{attribute 'qualified_only'}
VAR_GLOBAL
	bSWGreen 	AT%Q*	:BOOL;
	bSWRed 		AT%Q*	:BOOL;
END_VAR

(* stored: Version 1.1.0.1, ProductVersion 3.1.4026.6
   GVL Indicator: Id {c911d81c-9b6c-46b3-afa3-f72b033b7f4d} *)
